(* PLC project CoDeSys External Library Template, WAGO e!COCKPIT e!COCKPIT, author 3S - Smart Software Solutions GmbH *)
(* stored: creationDateTime 2019-10-29T12:37:19.490572, version 3.5.5.30, modificationDateTime 2019-10-29T12:36:39.3744516, organization 3S - Smart Software Solutions GmbH *)
(* Library project template with all possible element types, docu and a sample project structure *)

(* values of enumPPPSZadajnikTrybPracy: Manualny: Tryb pracy ręcznej; Automatyczny: Tryb pracy automatyczny *)

(* Autor: Paweł Kąkol, 2018-09-10-PK Prawa majątkowe: Solwena Sp. z o.o., Aktualizacje: 2018-10-02 - AW - Zmiana numeracji. Tryb Manualny na 0 2018-10-15 - AW - Zmiana numeracji. Dodanie trybów AutonomizacjaManualny i AutonomizacjaAutomatyczny 2018-12-12 - JB - Ujednolicenie trybów z siłownikiem SAB+. 2019-06-06 - AWy - Usunięcie trybów Wylaczenie, AutonomizacjaManualny i AutonomizacjaAutomatyczny oraz zmiana nazwy trybu Regulacja IZE na Automatyczny Opis: enum służy do obsługi Trybów pracy fb zadajnika SR04P (FCP0) na budynkach PPP Sopot (ENGIE) *)
{attribute 'qualified_only'}
{attribute 'strict'}
TYPE enumPPPSZadajnikTrybPracy : (Manualny := 0, Automatyczny := 1);
END_TYPE
